// TwinCAT 3 PLC project Main
// ProgramVersion: 3.1.4023.0
// libraries:
//   Tc2_Standard, * (Beckhoff Automation GmbH)
//   Tc2_System, * (Beckhoff Automation GmbH)
//   Tc3_Module, * (Beckhoff Automation GmbH)
// project tree:
//   DUTs/ MyStructure.TcDUT
//   GVLs/ GVL.TcGVL
//   / PlcTask.TcTTO
//   POUs/ MAIN.TcPOU
// real-time tasks:
//   TASK PlcTask: cycle T#10ms, priority 20, ADS port 350

CONFIGURATION Main
    RESOURCE PLC ON TwinCAT3
        TASK PlcTask(INTERVAL := T#10ms, PRIORITY := 20);
        PROGRAM MAIN WITH PlcTask : MAIN;
    END_RESOURCE
END_CONFIGURATION

// ---- DUTs/MyStructure.TcDUT
TYPE MyStructure :
STRUCT
	Name : STRING;
	Parameter_01 : REAL;
	Parameter_02 : REAL;
	Parameter_03 : REAL;
	Parameter_04 : REAL;
	Parameter_05 : REAL;
	Parameter_06 : REAL;
	Parameter_07 : REAL;
	Parameter_08 : REAL;
	Parameter_09 : REAL;
	Parameter_10 : REAL;
	Status : BOOL ;	
END_STRUCT
END_TYPE

// ---- GVLs/GVL.TcGVL
{attribute 'qualified_only'}
VAR_GLOBAL
	
	myArray : ARRAY [0..10] OF MyStructure;
	
END_VAR

// ---- POUs/MAIN.TcPOU
PROGRAM MAIN
VAR
END_VAR

END_PROGRAM
